{attribute 'linkalways'} 
{attribute 'no_explicit_call' := 'This FB is a CLASS and must be accessed using methods or properties'}
{attribute 'enable_dynamic_creation'}
FUNCTION_BLOCK Node_ContainerType_Vector_LREAL EXTENDS Node
VAR
    out : _GUID;
END_VAR

METHOD PUBLIC  Clone : I_Node
VAR
	pNode : POINTER TO Node_ContainerType_Vector_LREAL;
END_VAR
pNode := __NEW(Node_ContainerType_Vector_LREAL);
Clone := pNode^;
END_METHOD

METHOD FB_init : BOOL
VAR_INPUT
	bInitRetains : BOOL; // if TRUE, the retain variables are initialized (warm start / cold start)
	bInCopyCode : BOOL;  // if TRUE, the instance afterwards gets moved into the copy code (online change)
END_VAR
AddOutput('out', out);
END_METHOD

METHOD PROTECTED OnExecute
out.Value := ContainerType_Vector_LREAL;
END_METHOD

END_FUNCTION_BLOCK

(* stored: Version 1.1.0.1, ProductVersion 3.1.4026.17
   POU Node_ContainerType_Vector_LREAL: Id {3661a864-1763-0b39-039c-4cff9c5829f5}, SpecialFunc None
   Folder Constructor: Id {d86e404f-f63c-0f5c-16d9-4d740b85d3c4}
   Method Clone: Id {490d9b3e-fede-090f-3826-100d14cf8786}
   Method FB_init: Id {4fcc9fc6-ee8e-055b-2b50-bd93af9ef4a9}
   Method OnExecute: Id {f1817867-2834-09e9-171c-a993740a1a2c} *)
